% RSLogix 500 project AUTOMATIC DOOR_BAK006.RSS, saved by version 8.30.00.16 %
PROJECT "UNTITLED"    % processor: Bul.1763 MicroLogix 1100 Series B %

PROGRAM FILES
  LAD 2   6 rungs

DATA FILES
  O0 OUTPUT  4 elements
  I1 INPUT  6 elements
  S2 STATUS  66 elements
  B3 BINARY  1 elements
  T4 TIMER  1 elements
  C5 COUNTER  1 elements
  R6 CONTROL  1 elements
  N7 INTEGER  1 elements
  F8 FLOAT  1 elements

LADDER 2
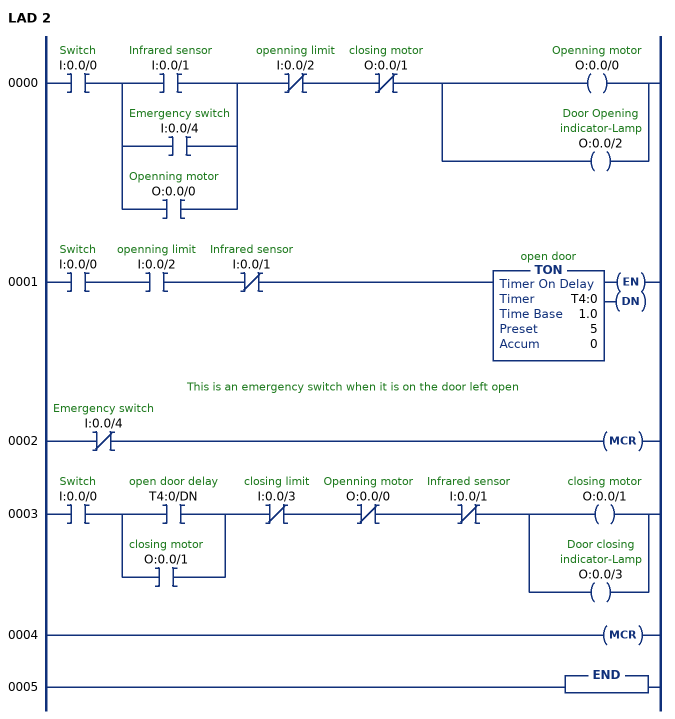
% Rung: 0 %
SOR XIC I:0.0/0 BST BST XIC I:0.0/1 NXB XIC I:0.0/4 BND NXB XIC O:0.0/0 BND XIO I:0.0/2 XIO O:0.0/1 BST OTE O:0.0/0 NXB OTE O:0.0/2 BND EOR
%   I:0.0/0  "Switch" %
%   I:0.0/1  "Infrared sensor" %
%   I:0.0/4  "Emergency switch" %
%   O:0.0/0  "Openning motor" %
%   I:0.0/2  "openning limit" %
%   O:0.0/1  "closing motor" %
%   O:0.0/2  "Door Opening indicator-Lamp" %
% Rung: 1 %
SOR XIC I:0.0/0 XIC I:0.0/2 XIO I:0.0/1 TON T4:0 1.0 5 0 EOR
%   I:0.0/0  "Switch" %
%   I:0.0/2  "openning limit" %
%   I:0.0/1  "Infrared sensor" %
%   T4:0  "open door" %
% Rung: 2 %
%                                                                  This is an emergency switch when it is on the door left open %
SOR XIO I:0.0/4 MCR EOR
%   I:0.0/4  "Emergency switch" %
% Rung: 3 %
SOR XIC I:0.0/0 BST XIC T4:0/DN NXB XIC O:0.0/1 BND XIO I:0.0/3 XIO O:0.0/0 XIO I:0.0/1 BST OTE O:0.0/1 NXB OTE O:0.0/3 BND EOR
%   I:0.0/0  "Switch" %
%   T4:0/DN  "open door delay" %
%   O:0.0/1  "closing motor" %
%   I:0.0/3  "closing limit" %
%   O:0.0/0  "Openning motor" %
%   I:0.0/1  "Infrared sensor" %
%   O:0.0/3  "Door closing indicator-Lamp" %
% Rung: 4 %
SOR MCR EOR
% Rung: 5 %
SOR END EOR

DATA TABLE (non-zero values as saved)
DATA T4
% .PRE .ACC %
% T4:0 % 5 0
